FUNCTION_BLOCK OFFSET_UDINT (* Take a first-Event Offset. *)
  (* Standard: 61499-1; Description: Copyright (c) 2024 HR Agrartechnik GmbH This program and the accompanying materials are made available under the terms of the Eclipse Public License 2.0 which is available at https://www.eclipse.org/legal/epl-2.0/ SPDX-License-Identifier: EPL-2.0 *)
  (* Version 1.0, 2024-10-18, Franz Höpfinger, HR Agrartechnik GmbH *)
  PACKAGE logiBUS::utils::math;
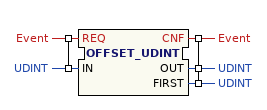
  EVENT_INPUT
    REQ WITH IN; (* Normal Execution Request *)
  END_EVENT
  EVENT_OUTPUT
    CNF WITH OUT, FIRST; (* Execution Confirmation *)
  END_EVENT
  VAR_INPUT
    IN : UDINT := 0; (* Input. First call with a Value >0 will Set FIRST *)
  END_VAR
  VAR_OUTPUT
    OUT : UDINT := 0; (* IN - FIRST *)
    FIRST : UDINT := 0; (* Set at First Call *)
  END_VAR
  EC_STATES
    REQ : REQ -> CNF;
  END_STATES
  ALGORITHM REQ IN ST:
IF (FIRST = 0) THEN
	FIRST := IN;
END_IF;

OUT := IN - FIRST;
  END_ALGORITHM
END_FUNCTION_BLOCK
